KUKA KRL program: chk_w5_wechs_ok.src

&ACCESS RVO7
&COMMENT Check Gripper Axor
DEF chk_w5_wechs_ok( )

; VERIFICAÇÃO DE FERRAMENTA: GRIPPER AXOR

WAIT FOR (($IN[161]) AND ($IN[169]) AND ($IN[177]) AND ($IN[185]) AND (NOT $IN[193]) AND ($IN[219]))

END
